// TIA Portal V17 export
// export: Created 2022-03-12T16:05:21.451342Z, ExportSetting WithDefaults, DisplayName Totally Integrated Automation Portal, DisplayVersion V17, DisplayName TIA Portal Openness, DisplayVersion V17, DisplayName TIA Portal Version Control Interface, DisplayVersion V17, DisplayName STEP 7 Professional, DisplayVersion V17, DisplayName STEP 7 Safety, DisplayVersion V17, DisplayName WinCC Advanced / Unified PC, DisplayVersion V17
DATA_BLOCK "WarningCfg"   // DB31601
TITLE = CPG_WarningCfg
{ S7_Optimized_Access := 'TRUE' }
AUTHOR : tech.team.motioncontrol@siemens.com
FAMILY : CPG
VERSION : 1.0
// Support: tech.team.motioncontrol@siemens.com
// Fax: +49 (0) 9131/98-1297
// stored: AutoNumber true, DBAccessibleFromOPCUA true, DBAccessibleFromWebserver true, IsOnlyStoredInLoadMemory false, IsRetainMemResEnabled false, IsWriteProtectedInAS false, MemoryReserve 0
   VAR
      Event { ExternalAccessible := 'False'; ExternalVisible := 'False'; ExternalWritable := 'False'; S7_SetPoint := 'True'} : Array[0.."CPG_NO_OF_CFG_WARNINGS_UPPER_LIM"] of "CPG_typeEventCfg";
   END_VAR
BEGIN
   // Event[0] : Warning Test
   // Event[1] : Low Bottle Supply
   // Event[2] : Low Label Supply
   // Event[3] : Spare
   // Event[4] : Spare
   // Event[5] : Spare
   // Event[6] : Spare
   // Event[7] : Spare
   // Event[8] : Spare
   // Event[9] : Spare
   // Event[10] : Spare
   // Event[11] : Spare
   // Event[12] : Spare
   // Event[13] : Spare
   // Event[14] : Spare
   // Event[15] : Spare
   // Event[16] : Spare
   // Event[17] : Spare
   // Event[18] : Spare
   // Event[19] : Spare
   // Event[20] : Spare
   // Event[21] : Spare
   // Event[22] : Spare
   // Event[23] : Spare
   // Event[24] : Spare
   // Event[25] : Spare
   // Event[26] : Spare
   // Event[27] : Spare
   // Event[28] : Spare
   // Event[29] : Spare
   Event[0].ID := 0;
   Event[1].ID := 1;
   Event[2].ID := 2;
   Event[3].ID := 3;
   Event[4].ID := 4;
   Event[5].ID := 5;
   Event[6].ID := 6;
   Event[7].ID := 7;
   Event[8].ID := 8;
   Event[9].ID := 9;
   Event[10].ID := 10;
   Event[11].ID := 11;
   Event[12].ID := 12;
   Event[13].ID := 13;
   Event[14].ID := 14;
   Event[15].ID := 15;
   Event[16].ID := 16;
   Event[17].ID := 17;
   Event[18].ID := 18;
   Event[19].ID := 19;
   Event[20].ID := 20;
   Event[21].ID := 21;
   Event[22].ID := 22;
   Event[23].ID := 23;
   Event[24].ID := 24;
   Event[25].ID := 25;
   Event[26].ID := 26;
   Event[27].ID := 27;
   Event[28].ID := 28;
   Event[29].ID := 29;
   Event[0].message[0..1] := 'Warning Test';
   Event[0].message[2] := 'Los Warning Test';
   Event[1].message[0] := 'Low Bottle Supply';
   Event[1].message[1] := 'Flaschenzufuhr niedrig';
   Event[1].message[2] := 'Las Low Bottle Supply';
   Event[2].message[0] := 'Low Label Supply';
   Event[2].message[1] := 'Etikettenzufuhr niedrig';
   Event[2].message[2] := 'Las Low Label Supply';
   Event[3].message[0] := 'Spare';
   Event[3].message[1] := 'Reserve';
   Event[3].message[2] := 'Spare';
   Event[4].message[0] := 'Spare';
   Event[4].message[1] := 'Reserve';
   Event[4].message[2] := 'Spare';
   Event[5].message[0] := 'Spare';
   Event[5].message[1] := 'Reserve';
   Event[5].message[2] := 'Spare';
   Event[6].message[0] := 'Spare';
   Event[6].message[1] := 'Reserve';
   Event[6].message[2] := 'Spare';
   Event[7].message[0] := 'Spare';
   Event[7].message[1] := 'Reserve';
   Event[7].message[2] := 'Spare';
   Event[8].message[0] := 'Spare';
   Event[8].message[1] := 'Reserve';
   Event[8].message[2] := 'Spare';
   Event[9].message[0] := 'Spare';
   Event[9].message[1] := 'Reserve';
   Event[9].message[2] := 'Spare';
   Event[10].message[0] := 'Spare';
   Event[10].message[1] := 'Reserve';
   Event[10].message[2] := 'Spare';
   Event[11].message[0] := 'Spare';
   Event[11].message[1] := 'Reserve';
   Event[11].message[2] := 'Spare';
   Event[12].message[0] := 'Spare';
   Event[12].message[1] := 'Reserve';
   Event[12].message[2] := 'Spare';
   Event[13].message[0] := 'Spare';
   Event[13].message[1] := 'Reserve';
   Event[13].message[2] := 'Spare';
   Event[14].message[0] := 'Spare';
   Event[14].message[1] := 'Reserve';
   Event[14].message[2] := 'Spare';
   Event[15].message[0] := 'Spare';
   Event[15].message[1] := 'Reserve';
   Event[15].message[2] := 'Spare';
   Event[16].message[0] := 'Spare';
   Event[16].message[1] := 'Reserve';
   Event[16].message[2] := 'Spare';
   Event[17].message[0] := 'Spare';
   Event[17].message[1] := 'Reserve';
   Event[17].message[2] := 'Spare';
   Event[18].message[0] := 'Spare';
   Event[18].message[1] := 'Reserve';
   Event[18].message[2] := 'Spare';
   Event[19].message[0] := 'Spare';
   Event[19].message[1] := 'Reserve';
   Event[19].message[2] := 'Spare';
   Event[20].message[0] := 'Spare';
   Event[20].message[1] := 'Reserve';
   Event[20].message[2] := 'Spare';
   Event[21].message[0] := 'Spare';
   Event[21].message[1] := 'Reserve';
   Event[21].message[2] := 'Spare';
   Event[22].message[0] := 'Spare';
   Event[22].message[1] := 'Reserve';
   Event[22].message[2] := 'Spare';
   Event[23].message[0] := 'Spare';
   Event[23].message[1] := 'Reserve';
   Event[23].message[2] := 'Spare';
   Event[24].message[0] := 'Spare';
   Event[24].message[1] := 'Reserve';
   Event[24].message[2] := 'Spare';
   Event[25].message[0] := 'Spare';
   Event[25].message[1] := 'Reserve';
   Event[25].message[2] := 'Spare';
   Event[26].message[0] := 'Spare';
   Event[26].message[1] := 'Reserve';
   Event[26].message[2] := 'Spare';
   Event[27].message[0] := 'Spare';
   Event[27].message[1] := 'Reserve';
   Event[27].message[2] := 'Spare';
   Event[28].message[0] := 'Spare';
   Event[28].message[1] := 'Reserve';
   Event[28].message[2] := 'Spare';
   Event[29].message[0] := 'Spare';
   Event[29].message[1] := 'Reserve';
   Event[29].message[2] := 'Spare';
END_DATA_BLOCK
